INTERFACE ITF_BaseExecutiveElement_HMI

END_INTERFACE

(* stored: Version 1.1.0.1
   Itf ITF_BaseExecutiveElement_HMI: Id {281655a4-c184-0338-36d1-b2c06941dfb5} *)
